FUNCTION_BLOCK fb_Station_LinkedList IMPLEMENTS I_Station_LinkedList
VAR
  _LastNodeAdded,
  _LastNodeRemoved  : ST_STATION_LIST_RESULT;

	_nCount           : UDINT;
  _nFree            : UDINT;

  {attribute 'hide'}
	_stList           : ARRAY[0..MAX_LIST_NODES] OF ST_STATION_MOVER_DATA;
	_stNodes          : ARRAY[0..MAX_LIST_NODES] OF T_LinkedListEntry;

	_fbList           : Tc2_Utilities.FB_LinkedListCtrl;
	_hList            : Tc2_Utilities.T_HLINKEDLIST;

	_stRef            : POINTER TO ST_STATION_MOVER_DATA;
END_VAR

METHOD AddHeadValue : ST_STATION_LIST_RESULT
VAR_INPUT
  stData        : ST_STATION_MOVER_DATA;
END_VAR
VAR
  _nIdxNode     : ULINT; 
	_pPosGet      : POINTER TO T_LinkedListEntry;
  _stRes        : ST_STATION_LIST_RESULT;
END_VAR

// add empty node
_fbList.A_AddHeadValue( hList     := _hList, 
                        putValue  := 16#0, 
                        getPosPtr => _pPosGet);

IF NOT _fbList.bOk 
THEN
  _stRes.wState.0       := TRUE;
ELSE
  // Get array index of new node
	_fbList.A_GetIndexAtPosPtr( hList       := _hList, 
                              putPosPtr   := _pPosGet, 
                              getValue    => _nIdxNode);

	IF NOT _fbList.bOk 
  THEN
    _stRes.wState.1     := TRUE;
  ELSE
    // write data to new node index
		_stRef 	            := ADR( _stList[_nIdxNode] );
		_stRef^ 	          := stData;

		_fbList.A_SetValueAtPosPtr( hList     := _hList, 
                                putPosPtr := _pPosGet, 
                                putValue  := _stRef);

		IF NOT _fbList.bOk 
    THEN
      _stRes.wState.2   := TRUE;
    ELSE
      _stRes.nIndex     := _nIdxNode;
			_stRes.stData     := stData;
      _LastNodeAdded    := _stRes;
		END_IF
	END_IF
END_IF

AddHeadValue := _stRes;
END_METHOD

METHOD AddTailValue : ST_STATION_LIST_RESULT
VAR_INPUT
  stData        : ST_STATION_MOVER_DATA;
END_VAR
VAR
  _nIdxNode     : ULINT; 
	_pPosGet      : POINTER TO T_LinkedListEntry;
  _stRes        : ST_STATION_LIST_RESULT;
END_VAR

// add empty node
_fbList.A_AddTailValue( hList       := _hList, 
                        putValue    := 16#0, 
                        getPosPtr   => _pPosGet);


IF NOT _fbList.bOk 
THEN
  _stRes.wState.0 := TRUE;
ELSE
  // Get array index of new node
	_fbList.A_GetIndexAtPosPtr( hList       := _hList, 
                              putPosPtr   := _pPosGet, 
                              getValue    => _nIdxNode);

	IF NOT _fbList.bOk 
  THEN
    _stRes.wState.1     := TRUE;
  ELSE
    // write data to new node index
		_stRef 	            := ADR( _stList[_nIdxNode] );
		_stRef^ 	          := stData;

		_fbList.A_SetValueAtPosPtr( hList     := _hList, 
                                putPosPtr := _pPosGet, 
                                putValue  := _stRef);

		IF NOT _fbList.bOk 
    THEN
      _stRes.wState.2   := TRUE;
    ELSE
      _stRes.nIndex     := _nIdxNode;
			_stRes.stData     := stData;
      _LastNodeAdded    := _stRes;
		END_IF
	END_IF
END_IF

AddTailValue := _stRes;
END_METHOD

PROPERTY Count : UDINT
GET
Count := _nCount := _hList.nCount;
END_GET
END_PROPERTY

PROPERTY Data : ARRAY[1..MAX_LIST_NODES] OF ST_STATION_MOVER_DATA
GET
VAR
	_tList        : ARRAY[1..MAX_LIST_NODES] OF ST_STATION_MOVER_DATA;
  _getValue     : PVOID;
  _pEntry       : POINTER TO ST_STATION_MOVER_DATA;
  _getPosPtr    : POINTER TO T_LinkedListEntry := 0;
  _nIdx         : UINT;  
END_VAR
_fbList(
	hList       := _hList);

_nCount       := _hList.nCount;
_nFree        := _hList.nFree;


_fbList.A_GetHead( hList := _hList, getValue=> _getValue, getPosPtr=> _getPosPtr );
IF _fbList.bOk 
THEN
  IF (_hList.nCount > 0)
  THEN
    _nIdx         := 1;
    _pEntry       := _getValue;
    _tList[1]     := _pEntry^;
    
    REPEAT
      _fbList.A_GetNext( hList := _hList, putPosPtr := _getPosPtr, getValue=> _getValue, getPosPtr=> _getPosPtr );
  
      IF _fbList.bOk THEN
        _nIdx         := _nIdx + 1;
        _pEntry       := _getValue;
        _tList[_nIdx] := _pEntry^;
      ELSE
        EXIT;
      END_IF
    UNTIL NOT _fbList.bOk
    END_REPEAT
  END_IF
END_IF

Data := _tList;
END_GET
END_PROPERTY

PROPERTY Free : UDINT
GET
Free := _nFree := _hList.nFree;
END_GET
END_PROPERTY

METHOD GetHead : ST_STATION_LIST_RESULT
VAR_INPUT
END_VAR
VAR
	_pPosGet      : POINTER TO T_LinkedListEntry;
  _pData        : POINTER TO ST_STATION_MOVER_DATA;
  _stRes        : ST_STATION_LIST_RESULT;
END_VAR

_fbList.A_GetHead(hList      := _hList,
                  getValue   => _pData,
                  getPosPtr  => _pPosGet);

IF NOT _fbList.bOk
THEN
  _stRes.wState.0 := TRUE;
ELSE
  _stRes.stData := _pData^;
END_IF

GetHead := _stRes;
END_METHOD

METHOD GetTail : ST_STATION_LIST_RESULT
VAR_INPUT
END_VAR
VAR
	_pPosGet      : POINTER TO T_LinkedListEntry;
  _pData        : POINTER TO ST_STATION_MOVER_DATA;
  _stRes        : ST_STATION_LIST_RESULT;
END_VAR

_fbList.A_GetTail(hList      := _hList,
                  getValue   => _pData,
                  getPosPtr  => _pPosGet);

IF NOT _fbList.bOk
THEN
  _stRes.wState.0 := TRUE;
ELSE
  _stRes.stData := _pData^;
END_IF

GetTail := _stRes;
END_METHOD

METHOD InitList : BOOL
VAR
  _bOk : Bool;
END_VAR

IF Tc2_Utilities.F_CreateLinkedListHnd(ADR(_stNodes), SIZEOF(_stNodes), _hList)
THEN
  _fbList.A_Reset(hList := _hList, bOk => _bOk);
  memset(ADR(_stList), 0, SIZEOF(_stList));
  _nCount   := 0;
  InitList  := TRUE; //_bOk;
END_IF
END_METHOD

PROPERTY Nodes : ARRAY[0..MAX_LIST_NODES] OF T_LinkedListEntry
GET
Nodes := _stNodes;
END_GET
END_PROPERTY

METHOD RemoveHeadValue : ST_STATION_LIST_RESULT
VAR_INPUT
END_VAR
VAR
	_pPosGet      : POINTER TO T_LinkedListEntry;
  _pData        : POINTER TO ST_STATION_MOVER_DATA;
  _stRes        : ST_STATION_LIST_RESULT;
END_VAR
_fbList.A_RemoveHeadValue(hList       := _hList, 
                          getValue    => _pData, 
                          getPosPtr   => _pPosGet);

IF NOT _fbList.bOk 
THEN
  _stRes.wState.0 := TRUE;
ELSE
	_stRes.stData     := _pData^;
  _LastNodeRemoved  := _stRes;
  memset(_pData, 0, SIZEOF(ST_STATION_MOVER_DATA));
END_IF
RemoveHeadValue := _stRes;
END_METHOD

END_FUNCTION_BLOCK

(* stored: Version 1.1.0.1, ProductVersion 3.1.4026.13
   POU fb_Station_LinkedList: Id {f01f0db4-80d5-4efa-bc0e-a8532a3b5f97}, SpecialFunc None
   Method AddHeadValue: Id {dacf8335-e195-40f4-965e-7898f564145d}
   Method AddTailValue: Id {fc6a0a7f-f3d7-40bb-8cbf-5d716e2fd4c6}
   Property Count: Id {b519167c-e84b-4b4f-81ec-031dd682ef5b}
   Get Get: Id {eb31e2ef-23bc-4dba-b1b7-814df3cff826}
   Property Data: Id {876b4791-0fc6-425c-b5f8-389ba4c57541}
   Get Get: Id {0bfbe2e9-20ca-4718-91b7-a82533aef391}
   Property Free: Id {a07533ce-084a-4f80-85c4-f0df25b0adb1}
   Get Get: Id {f8d4dfc9-1cc8-45d8-8c9b-6c822c2f58ca}
   Method GetHead: Id {de72de40-01c2-4c26-aabf-0a7bf1751087}
   Method GetTail: Id {f6453a1a-87b8-4222-87d2-b9dde0aeaeb7}
   Method InitList: Id {177cbf3b-9097-415a-a37a-9ff40ae42c86}
   Property Nodes: Id {4b1c71a6-f6ed-4b43-b29e-54dda159e2d8}
   Get Get: Id {829f9d20-32a4-4c74-9a3e-0c4aeff09d55}
   Method RemoveHeadValue: Id {c9de05c0-b875-489a-a264-9b6b9d8d71fd} *)
